FUNCTION_BLOCK ATM_IN_MS_TO_AULI (* Convert TIME (via ATM adapter) in MS to ULINT (via AULI adapter) *)
  (* Standard: 61499-2; Description: Copyright (c) 2026 HR Agrartechnik GmbH This program and the accompanying materials are made available under the terms of the Eclipse Public License 2.0 which is available at https://www.eclipse.org/legal/epl-2.0/ SPDX-License-Identifier: EPL-2.0 *)
  (* Version 1.0, 2026-08-13, Franz Höpfinger, HR Agrartechnik GmbH, initial API and implementation *)
  PACKAGE adapter::conversion::unidirectional;
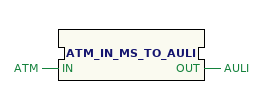
  SOCKETS
    IN : adapter::types::unidirectional::ATM; (* Time value to convert *)
  END_SOCKETS
  PLUGS
    OUT : adapter::types::unidirectional::AULI; (* TIME value of IN expressed in MS as ULINT *)
  END_PLUGS
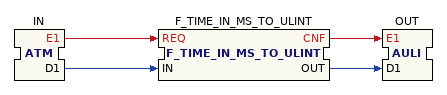
  FBS
    F_TIME_IN_MS_TO_ULINT : iec61131::conversion::F_TIME_IN_MS_TO_ULINT;
  END_FBS
  EVENT_CONNECTIONS
    IN.E1 TO F_TIME_IN_MS_TO_ULINT.REQ;
    F_TIME_IN_MS_TO_ULINT.CNF TO OUT.E1;
  END_CONNECTIONS
  DATA_CONNECTIONS
    IN.D1 TO F_TIME_IN_MS_TO_ULINT.IN;
    F_TIME_IN_MS_TO_ULINT.OUT TO OUT.D1;
  END_CONNECTIONS
END_FUNCTION_BLOCK
